PROGRAM Comp02_Sequencer
VAR
	ActiveStep 	: INT;
	Step1000	: Step;
	Step1100	: Step;
END_VAR

CASE Comp02.StateManager.oState OF
	State.Aborting:		Comp02_SeqAborting();
	State.Aborted:		Comp02_SeqAborted();
	State.Resetting:	Comp02_SeqResetting();
	State.Stopped:		Comp02_SeqStopped();
	State.Starting:		Comp02_SeqStarting();
	State.Running:		Comp02_SeqRunning();
	State.Pausing:		Comp02_SeqPausing();
	State.Paused:		Comp02_SeqPaused();
	State.Resuming:		Comp02_SeqResuming();
	State.Stopping:		Comp02_SeqStopping();	
END_CASE

ACTION Comp02_SeqAborted:

END_ACTION

ACTION Comp02_SeqAborting:

END_ACTION

ACTION Comp02_SeqPaused:

END_ACTION

ACTION Comp02_SeqPausing:

END_ACTION

ACTION Comp02_SeqResetting:

END_ACTION

ACTION Comp02_SeqResuming:

END_ACTION

ACTION Comp02_SeqRunning:
Step1000(	cDescription		:= 'Raise Blade Stop',
			cThisStep			:= 1000,
			cNextStep			:= 1100,
			cRecoveryStep		:= 1050,
			cTimeoutPreset 		:= T#5S,
			ioActiveStep 		:= ActiveStep);

IF Step1000.sActive THEN
			Comp01.D02_ACT1.iCmd	:= CmdActuator.Extend;
			Step1000.iComplete	:= TRUE;
END_IF			

//=============================================================================//
			
Step1100(	cDescription	:= 'Enable D06 Servo 1',
			cThisStep		:= 1100,
			cNextStep		:= 1200,
			cRecoveryStep	:= 1150,
			cTimeoutPreset 	:= T#5S,
			ioActiveStep 	:= ActiveStep);

IF Step1100.sActive THEN
			Comp01.PartLoader_Pusher.iCmd	:= CmdServo.Enable;
			Step1100.iComplete	:= TRUE;
END_IF		

//=============================================================================//
END_ACTION

ACTION Comp02_SeqStarting:

END_ACTION

ACTION Comp02_SeqStopped:

END_ACTION

ACTION Comp02_SeqStopping:

END_ACTION

END_PROGRAM

(* stored: Version 1.1.0.1, ProductVersion 3.1.4022.11
   POU Comp02_Sequencer: Id {54aa1706-180c-420d-9185-7238ffa35960}, SpecialFunc None
   Action Comp02_SeqAborted: Id {ecda4b35-a6f9-4aa4-9a0b-55ecbae06c4e}
   Action Comp02_SeqAborting: Id {12488e60-9902-4664-8e4c-60bafe664814}
   Action Comp02_SeqPaused: Id {34b4e2ba-2645-4e5b-8dce-a337f41cf9c3}
   Action Comp02_SeqPausing: Id {ea509241-fa55-4fc3-b8e3-92f4ce0ba158}
   Action Comp02_SeqResetting: Id {5c304fbd-47d2-454c-b058-6eba2db2b53a}
   Action Comp02_SeqResuming: Id {b970d7f8-8fa0-41d9-be91-2cbb1af3d079}
   Action Comp02_SeqRunning: Id {082ff177-30d7-495f-b4a2-182490cbe579}
   Action Comp02_SeqStarting: Id {e3f6040b-a1c5-4df7-99cd-ed5f58e20177}
   Action Comp02_SeqStopped: Id {8993345e-06a2-4b6a-bf5a-01e0cfdeceba}
   Action Comp02_SeqStopping: Id {d95151f3-038e-4a73-97ee-e2b4fc12893f} *)
